// TIA Portal V19 export
FUNCTION "RO_1" : Void   // FC10, LAD
{ S7_Optimized_Access := 'TRUE' }
// stored: SetENOAutomatically false
   VAR_TEMP   // added for the SCL form of the ladder/FBD networks
      _w1 : Bool;
      _w2 : Bool;
      _w3 : Bool;
   END_VAR
BEGIN

REGION Network 1: ABV-301/ ABV-302
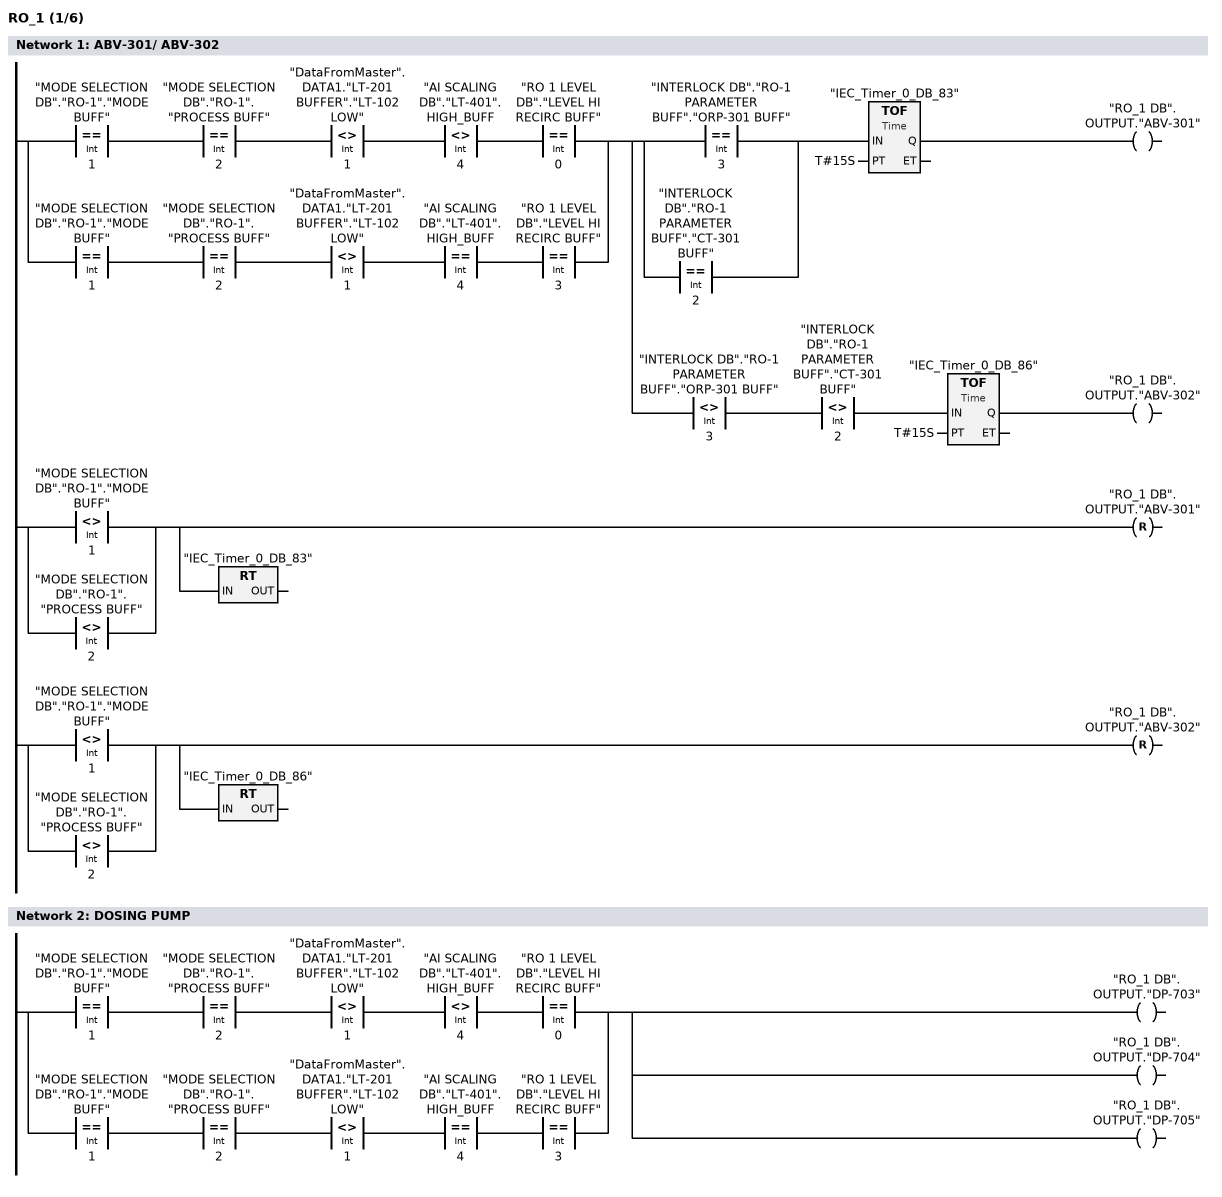
   RUNG wire#powerrail
      { S7_Templates := "SrcType := Int" } EQ_Contact(in1 := "MODE SELECTION DB"."RO-1"."MODE BUFF", in2 := 1)
      { S7_Templates := "SrcType := Int" } EQ_Contact(in1 := "MODE SELECTION DB"."RO-1"."PROCESS BUFF", in2 := 2)
      { S7_Templates := "SrcType := Int" } NE_Contact(in1 := "DataFromMaster".DATA1."LT-201 BUFFER"."LT-102 LOW", in2 := 1)
      { S7_Templates := "SrcType := Int" } NE_Contact(in1 := "AI SCALING DB"."LT-401".HIGH_BUFF, in2 := 4)
      { S7_Templates := "SrcType := Int" } EQ_Contact(in1 := "RO 1 LEVEL DB"."LEVEL HI RECIRC BUFF", in2 := 0)
      wire#w1
      { S7_Templates := "SrcType := Int" } EQ_Contact(in1 := "INTERLOCK DB"."RO-1 PARAMETER BUFF"."ORP-301 BUFF", in2 := 3)
      wire#w2
      { S7_Templates := "time_type := Time" } "IEC_Timer_0_DB_83".TOF(pt := T#15S, et =>)
      Coil( "RO_1 DB".OUTPUT."ABV-301" )
   END_RUNG
   RUNG wire#powerrail
      { S7_Templates := "SrcType := Int" } EQ_Contact(in1 := "MODE SELECTION DB"."RO-1"."MODE BUFF", in2 := 1)
      { S7_Templates := "SrcType := Int" } EQ_Contact(in1 := "MODE SELECTION DB"."RO-1"."PROCESS BUFF", in2 := 2)
      { S7_Templates := "SrcType := Int" } NE_Contact(in1 := "DataFromMaster".DATA1."LT-201 BUFFER"."LT-102 LOW", in2 := 1)
      { S7_Templates := "SrcType := Int" } EQ_Contact(in1 := "AI SCALING DB"."LT-401".HIGH_BUFF, in2 := 4)
      { S7_Templates := "SrcType := Int" } EQ_Contact(in1 := "RO 1 LEVEL DB"."LEVEL HI RECIRC BUFF", in2 := 3)
   END_RUNG wire#w1
   RUNG wire#w1
      { S7_Templates := "SrcType := Int" } EQ_Contact(in1 := "INTERLOCK DB"."RO-1 PARAMETER BUFF"."CT-301 BUFF", in2 := 2)
   END_RUNG wire#w2
   RUNG wire#w1
      { S7_Templates := "SrcType := Int" } NE_Contact(in1 := "INTERLOCK DB"."RO-1 PARAMETER BUFF"."ORP-301 BUFF", in2 := 3)
      { S7_Templates := "SrcType := Int" } NE_Contact(in1 := "INTERLOCK DB"."RO-1 PARAMETER BUFF"."CT-301 BUFF", in2 := 2)
      { S7_Templates := "time_type := Time" } "IEC_Timer_0_DB_86".TOF(pt := T#15S, et =>)
      Coil( "RO_1 DB".OUTPUT."ABV-302" )
   END_RUNG
   RUNG wire#powerrail
      { S7_Templates := "SrcType := Int" } NE_Contact(in1 := "MODE SELECTION DB"."RO-1"."MODE BUFF", in2 := 1)
      wire#w3
      R_Coil( "RO_1 DB".OUTPUT."ABV-301" )
   END_RUNG
   RUNG wire#powerrail
      { S7_Templates := "SrcType := Int" } NE_Contact(in1 := "MODE SELECTION DB"."RO-1"."PROCESS BUFF", in2 := 2)
   END_RUNG wire#w3
   RUNG wire#w3
      RT_Coil( "IEC_Timer_0_DB_83" )
   END_RUNG
   RUNG wire#powerrail
      { S7_Templates := "SrcType := Int" } NE_Contact(in1 := "MODE SELECTION DB"."RO-1"."MODE BUFF", in2 := 1)
      wire#w4
      R_Coil( "RO_1 DB".OUTPUT."ABV-302" )
   END_RUNG
   RUNG wire#powerrail
      { S7_Templates := "SrcType := Int" } NE_Contact(in1 := "MODE SELECTION DB"."RO-1"."PROCESS BUFF", in2 := 2)
   END_RUNG wire#w4
   RUNG wire#w4
      RT_Coil( "IEC_Timer_0_DB_86" )
   END_RUNG
   // the same network as SCL:
   #_w1 := (("MODE SELECTION DB"."RO-1"."MODE BUFF" = 1) AND ("MODE SELECTION DB"."RO-1"."PROCESS BUFF" = 2) AND ("DataFromMaster".DATA1."LT-201 BUFFER"."LT-102 LOW" <> 1) AND ("AI SCALING DB"."LT-401".HIGH_BUFF <> 4) AND ("RO 1 LEVEL DB"."LEVEL HI RECIRC BUFF" = 0)) OR (("MODE SELECTION DB"."RO-1"."MODE BUFF" = 1) AND ("MODE SELECTION DB"."RO-1"."PROCESS BUFF" = 2) AND ("DataFromMaster".DATA1."LT-201 BUFFER"."LT-102 LOW" <> 1) AND ("AI SCALING DB"."LT-401".HIGH_BUFF = 4) AND ("RO 1 LEVEL DB"."LEVEL HI RECIRC BUFF" = 3));
   "IEC_Timer_0_DB_83".TOF(IN := #_w1 AND (("INTERLOCK DB"."RO-1 PARAMETER BUFF"."ORP-301 BUFF" = 3) OR ("INTERLOCK DB"."RO-1 PARAMETER BUFF"."CT-301 BUFF" = 2)),
                           PT := T#15S);
   "RO_1 DB".OUTPUT."ABV-301" := "IEC_Timer_0_DB_83".Q;
   "IEC_Timer_0_DB_86".TOF(IN := #_w1 AND ("INTERLOCK DB"."RO-1 PARAMETER BUFF"."ORP-301 BUFF" <> 3) AND ("INTERLOCK DB"."RO-1 PARAMETER BUFF"."CT-301 BUFF" <> 2),
                           PT := T#15S);
   "RO_1 DB".OUTPUT."ABV-302" := "IEC_Timer_0_DB_86".Q;
   #_w2 := ("MODE SELECTION DB"."RO-1"."MODE BUFF" <> 1) OR ("MODE SELECTION DB"."RO-1"."PROCESS BUFF" <> 2);
   IF #_w2 THEN
       "RO_1 DB".OUTPUT."ABV-301" := FALSE;
       RESET_TIMER("IEC_Timer_0_DB_83");
   END_IF;
   #_w3 := ("MODE SELECTION DB"."RO-1"."MODE BUFF" <> 1) OR ("MODE SELECTION DB"."RO-1"."PROCESS BUFF" <> 2);
   IF #_w3 THEN
       "RO_1 DB".OUTPUT."ABV-302" := FALSE;
       RESET_TIMER("IEC_Timer_0_DB_86");
   END_IF;
END_REGION

REGION Network 2: DOSING PUMP
   RUNG wire#powerrail
      { S7_Templates := "SrcType := Int" } EQ_Contact(in1 := "MODE SELECTION DB"."RO-1"."MODE BUFF", in2 := 1)
      { S7_Templates := "SrcType := Int" } EQ_Contact(in1 := "MODE SELECTION DB"."RO-1"."PROCESS BUFF", in2 := 2)
      { S7_Templates := "SrcType := Int" } NE_Contact(in1 := "DataFromMaster".DATA1."LT-201 BUFFER"."LT-102 LOW", in2 := 1)
      { S7_Templates := "SrcType := Int" } NE_Contact(in1 := "AI SCALING DB"."LT-401".HIGH_BUFF, in2 := 4)
      { S7_Templates := "SrcType := Int" } EQ_Contact(in1 := "RO 1 LEVEL DB"."LEVEL HI RECIRC BUFF", in2 := 0)
      wire#w1
      Coil( "RO_1 DB".OUTPUT."DP-703" )
   END_RUNG
   RUNG wire#powerrail
      { S7_Templates := "SrcType := Int" } EQ_Contact(in1 := "MODE SELECTION DB"."RO-1"."MODE BUFF", in2 := 1)
      { S7_Templates := "SrcType := Int" } EQ_Contact(in1 := "MODE SELECTION DB"."RO-1"."PROCESS BUFF", in2 := 2)
      { S7_Templates := "SrcType := Int" } NE_Contact(in1 := "DataFromMaster".DATA1."LT-201 BUFFER"."LT-102 LOW", in2 := 1)
      { S7_Templates := "SrcType := Int" } EQ_Contact(in1 := "AI SCALING DB"."LT-401".HIGH_BUFF, in2 := 4)
      { S7_Templates := "SrcType := Int" } EQ_Contact(in1 := "RO 1 LEVEL DB"."LEVEL HI RECIRC BUFF", in2 := 3)
   END_RUNG wire#w1
   RUNG wire#w1
      Coil( "RO_1 DB".OUTPUT."DP-704" )
   END_RUNG
   RUNG wire#w1
      Coil( "RO_1 DB".OUTPUT."DP-705" )
   END_RUNG
   // the same network as SCL:
   "RO_1 DB".OUTPUT."DP-703" := (("MODE SELECTION DB"."RO-1"."MODE BUFF" = 1) AND ("MODE SELECTION DB"."RO-1"."PROCESS BUFF" = 2) AND ("DataFromMaster".DATA1."LT-201 BUFFER"."LT-102 LOW" <> 1) AND ("AI SCALING DB"."LT-401".HIGH_BUFF <> 4) AND ("RO 1 LEVEL DB"."LEVEL HI RECIRC BUFF" = 0)) OR (("MODE SELECTION DB"."RO-1"."MODE BUFF" = 1) AND ("MODE SELECTION DB"."RO-1"."PROCESS BUFF" = 2) AND ("DataFromMaster".DATA1."LT-201 BUFFER"."LT-102 LOW" <> 1) AND ("AI SCALING DB"."LT-401".HIGH_BUFF = 4) AND ("RO 1 LEVEL DB"."LEVEL HI RECIRC BUFF" = 3));
   "RO_1 DB".OUTPUT."DP-704" := "RO_1 DB".OUTPUT."DP-703";
   "RO_1 DB".OUTPUT."DP-705" := "RO_1 DB".OUTPUT."DP-703";
END_REGION

REGION Network 3: RO-1 FEED PUMP
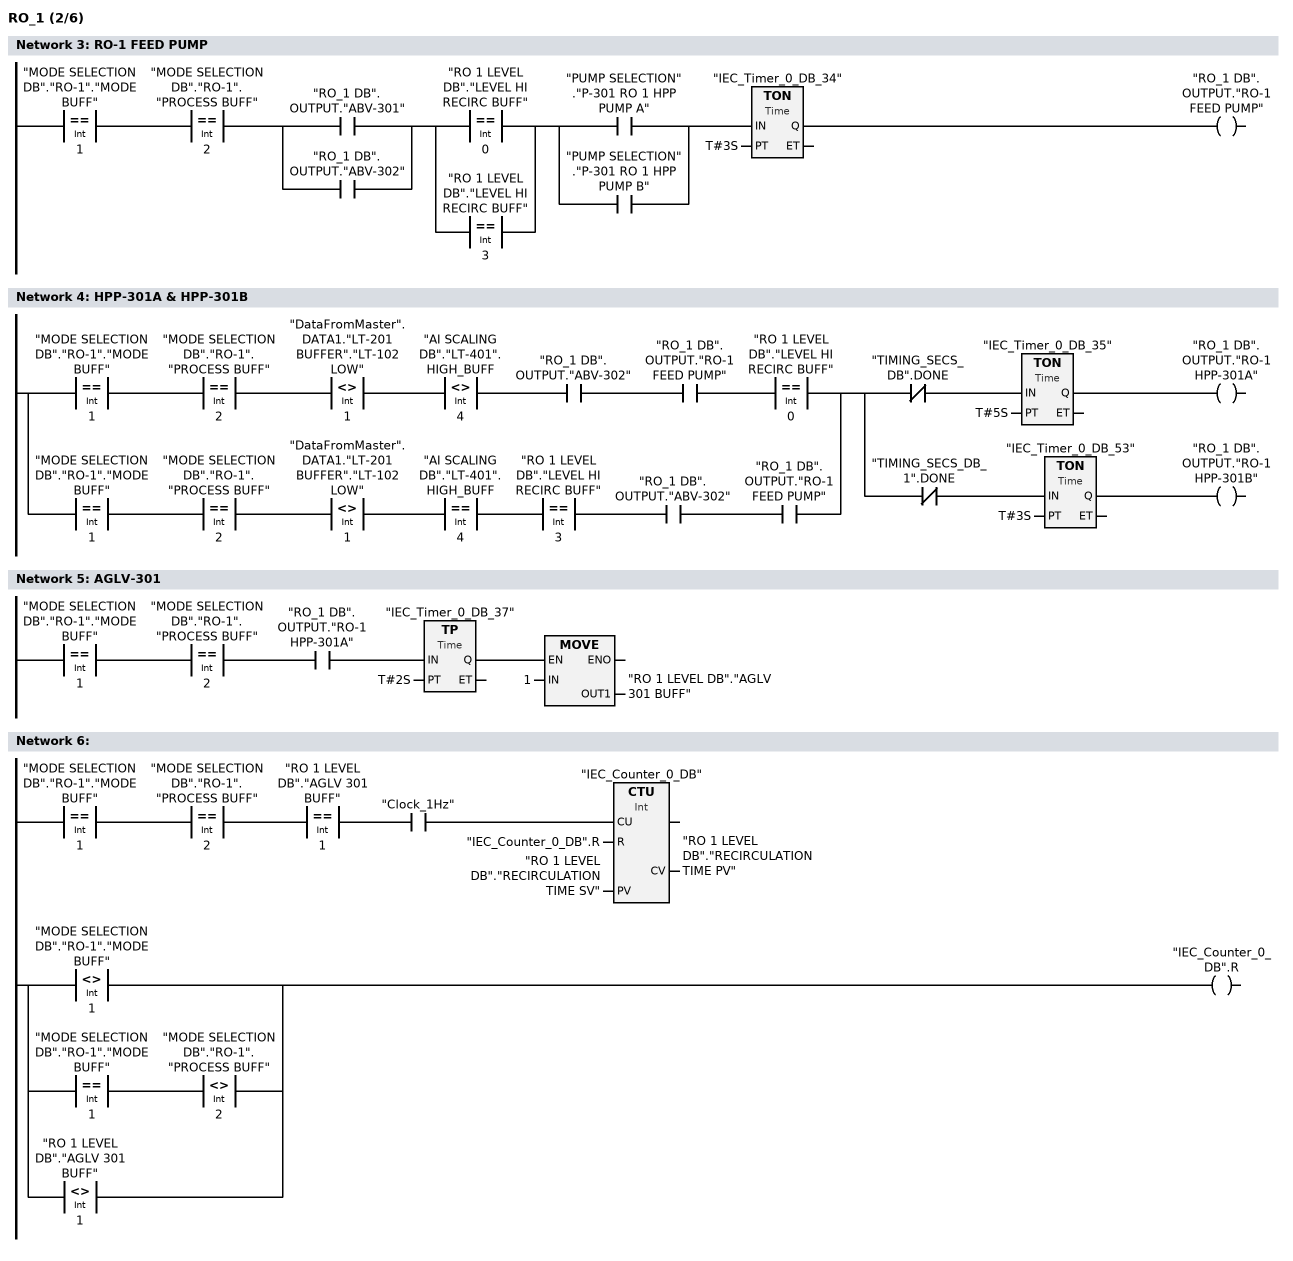
   RUNG wire#powerrail
      { S7_Templates := "SrcType := Int" } EQ_Contact(in1 := "MODE SELECTION DB"."RO-1"."MODE BUFF", in2 := 1)
      { S7_Templates := "SrcType := Int" } EQ_Contact(in1 := "MODE SELECTION DB"."RO-1"."PROCESS BUFF", in2 := 2)
      wire#w1
      Contact( "RO_1 DB".OUTPUT."ABV-301" )
      wire#w2
      { S7_Templates := "SrcType := Int" } EQ_Contact(in1 := "RO 1 LEVEL DB"."LEVEL HI RECIRC BUFF", in2 := 0)
      wire#w3
      Contact( "PUMP SELECTION"."P-301 RO 1 HPP PUMP A" )
      wire#w4
      { S7_Templates := "time_type := Time" } "IEC_Timer_0_DB_34".TON(pt := T#3S, et =>)
      Coil( "RO_1 DB".OUTPUT."RO-1 FEED PUMP" )
   END_RUNG
   RUNG wire#w1
      Contact( "RO_1 DB".OUTPUT."ABV-302" )
   END_RUNG wire#w2
   RUNG wire#w2
      { S7_Templates := "SrcType := Int" } EQ_Contact(in1 := "RO 1 LEVEL DB"."LEVEL HI RECIRC BUFF", in2 := 3)
   END_RUNG wire#w3
   RUNG wire#w3
      Contact( "PUMP SELECTION"."P-301 RO 1 HPP PUMP B" )
   END_RUNG wire#w4
   // the same network as SCL:
   "IEC_Timer_0_DB_34".TON(IN := ("MODE SELECTION DB"."RO-1"."MODE BUFF" = 1) AND ("MODE SELECTION DB"."RO-1"."PROCESS BUFF" = 2) AND ("RO_1 DB".OUTPUT."ABV-301" OR "RO_1 DB".OUTPUT."ABV-302") AND (("RO 1 LEVEL DB"."LEVEL HI RECIRC BUFF" = 0) OR ("RO 1 LEVEL DB"."LEVEL HI RECIRC BUFF" = 3)) AND ("PUMP SELECTION"."P-301 RO 1 HPP PUMP A" OR "PUMP SELECTION"."P-301 RO 1 HPP PUMP B"),
                           PT := T#3S);
   "RO_1 DB".OUTPUT."RO-1 FEED PUMP" := "IEC_Timer_0_DB_34".Q;
END_REGION

REGION Network 4: HPP-301A & HPP-301B
   RUNG wire#powerrail
      { S7_Templates := "SrcType := Int" } EQ_Contact(in1 := "MODE SELECTION DB"."RO-1"."MODE BUFF", in2 := 1)
      { S7_Templates := "SrcType := Int" } EQ_Contact(in1 := "MODE SELECTION DB"."RO-1"."PROCESS BUFF", in2 := 2)
      { S7_Templates := "SrcType := Int" } NE_Contact(in1 := "DataFromMaster".DATA1."LT-201 BUFFER"."LT-102 LOW", in2 := 1)
      { S7_Templates := "SrcType := Int" } NE_Contact(in1 := "AI SCALING DB"."LT-401".HIGH_BUFF, in2 := 4)
      Contact( "RO_1 DB".OUTPUT."ABV-302" )
      Contact( "RO_1 DB".OUTPUT."RO-1 FEED PUMP" )
      { S7_Templates := "SrcType := Int" } EQ_Contact(in1 := "RO 1 LEVEL DB"."LEVEL HI RECIRC BUFF", in2 := 0)
      wire#w1
      I_Contact( "TIMING_SECS_DB".DONE )
      { S7_Templates := "time_type := Time" } "IEC_Timer_0_DB_35".TON(pt := T#5S, et =>)
      Coil( "RO_1 DB".OUTPUT."RO-1 HPP-301A" )
   END_RUNG
   RUNG wire#powerrail
      { S7_Templates := "SrcType := Int" } EQ_Contact(in1 := "MODE SELECTION DB"."RO-1"."MODE BUFF", in2 := 1)
      { S7_Templates := "SrcType := Int" } EQ_Contact(in1 := "MODE SELECTION DB"."RO-1"."PROCESS BUFF", in2 := 2)
      { S7_Templates := "SrcType := Int" } NE_Contact(in1 := "DataFromMaster".DATA1."LT-201 BUFFER"."LT-102 LOW", in2 := 1)
      { S7_Templates := "SrcType := Int" } EQ_Contact(in1 := "AI SCALING DB"."LT-401".HIGH_BUFF, in2 := 4)
      { S7_Templates := "SrcType := Int" } EQ_Contact(in1 := "RO 1 LEVEL DB"."LEVEL HI RECIRC BUFF", in2 := 3)
      Contact( "RO_1 DB".OUTPUT."ABV-302" )
      Contact( "RO_1 DB".OUTPUT."RO-1 FEED PUMP" )
   END_RUNG wire#w1
   RUNG wire#w1
      I_Contact( "TIMING_SECS_DB_1".DONE )
      { S7_Templates := "time_type := Time" } "IEC_Timer_0_DB_53".TON(pt := T#3S, et =>)
      Coil( "RO_1 DB".OUTPUT."RO-1 HPP-301B" )
   END_RUNG
   // the same network as SCL:
   #_w1 := (("MODE SELECTION DB"."RO-1"."MODE BUFF" = 1) AND ("MODE SELECTION DB"."RO-1"."PROCESS BUFF" = 2) AND ("DataFromMaster".DATA1."LT-201 BUFFER"."LT-102 LOW" <> 1) AND ("AI SCALING DB"."LT-401".HIGH_BUFF <> 4) AND "RO_1 DB".OUTPUT."ABV-302" AND "RO_1 DB".OUTPUT."RO-1 FEED PUMP" AND ("RO 1 LEVEL DB"."LEVEL HI RECIRC BUFF" = 0)) OR (("MODE SELECTION DB"."RO-1"."MODE BUFF" = 1) AND ("MODE SELECTION DB"."RO-1"."PROCESS BUFF" = 2) AND ("DataFromMaster".DATA1."LT-201 BUFFER"."LT-102 LOW" <> 1) AND ("AI SCALING DB"."LT-401".HIGH_BUFF = 4) AND ("RO 1 LEVEL DB"."LEVEL HI RECIRC BUFF" = 3) AND "RO_1 DB".OUTPUT."ABV-302" AND "RO_1 DB".OUTPUT."RO-1 FEED PUMP");
   "IEC_Timer_0_DB_35".TON(IN := #_w1 AND NOT "TIMING_SECS_DB".DONE, PT := T#5S);
   "RO_1 DB".OUTPUT."RO-1 HPP-301A" := "IEC_Timer_0_DB_35".Q;
   "IEC_Timer_0_DB_53".TON(IN := #_w1 AND NOT "TIMING_SECS_DB_1".DONE, PT := T#3S);
   "RO_1 DB".OUTPUT."RO-1 HPP-301B" := "IEC_Timer_0_DB_53".Q;
END_REGION

REGION Network 5: AGLV-301
   RUNG wire#powerrail
      { S7_Templates := "SrcType := Int" } EQ_Contact(in1 := "MODE SELECTION DB"."RO-1"."MODE BUFF", in2 := 1)
      { S7_Templates := "SrcType := Int" } EQ_Contact(in1 := "MODE SELECTION DB"."RO-1"."PROCESS BUFF", in2 := 2)
      Contact( "RO_1 DB".OUTPUT."RO-1 HPP-301A" )
      { S7_Templates := "time_type := Time" } "IEC_Timer_0_DB_37".TP(pt := T#2S, et =>)
      Move(in := 1, out1 => "RO 1 LEVEL DB"."AGLV 301 BUFF")
   END_RUNG
   // the same network as SCL:
   "IEC_Timer_0_DB_37".TP(IN := ("MODE SELECTION DB"."RO-1"."MODE BUFF" = 1) AND ("MODE SELECTION DB"."RO-1"."PROCESS BUFF" = 2) AND "RO_1 DB".OUTPUT."RO-1 HPP-301A",
                          PT := T#2S);
   IF "IEC_Timer_0_DB_37".Q THEN "RO 1 LEVEL DB"."AGLV 301 BUFF" := 1; END_IF;
END_REGION

REGION Network 6
   RUNG wire#powerrail
      { S7_Templates := "SrcType := Int" } EQ_Contact(in1 := "MODE SELECTION DB"."RO-1"."MODE BUFF", in2 := 1)
      { S7_Templates := "SrcType := Int" } EQ_Contact(in1 := "MODE SELECTION DB"."RO-1"."PROCESS BUFF", in2 := 2)
      { S7_Templates := "SrcType := Int" } EQ_Contact(in1 := "RO 1 LEVEL DB"."AGLV 301 BUFF", in2 := 1)
      Contact( "Clock_1Hz" )
      { S7_Templates := "value_type := Int" } "IEC_Counter_0_DB".CTU(r := "IEC_Counter_0_DB".R, pv := "RO 1 LEVEL DB"."RECIRCULATION TIME SV", cv => "RO 1 LEVEL DB"."RECIRCULATION TIME PV")
   END_RUNG
   RUNG wire#powerrail
      { S7_Templates := "SrcType := Int" } NE_Contact(in1 := "MODE SELECTION DB"."RO-1"."MODE BUFF", in2 := 1)
      wire#w1
      Coil( "IEC_Counter_0_DB".R )
   END_RUNG
   RUNG wire#powerrail
      { S7_Templates := "SrcType := Int" } EQ_Contact(in1 := "MODE SELECTION DB"."RO-1"."MODE BUFF", in2 := 1)
      { S7_Templates := "SrcType := Int" } NE_Contact(in1 := "MODE SELECTION DB"."RO-1"."PROCESS BUFF", in2 := 2)
   END_RUNG wire#w1
   RUNG wire#powerrail
      { S7_Templates := "SrcType := Int" } NE_Contact(in1 := "RO 1 LEVEL DB"."AGLV 301 BUFF", in2 := 1)
   END_RUNG wire#w1
   // the same network as SCL:
   "IEC_Counter_0_DB".CTU(CU := ("MODE SELECTION DB"."RO-1"."MODE BUFF" = 1) AND ("MODE SELECTION DB"."RO-1"."PROCESS BUFF" = 2) AND ("RO 1 LEVEL DB"."AGLV 301 BUFF" = 1) AND "Clock_1Hz",
                          R := "IEC_Counter_0_DB".R,
                          PV := "RO 1 LEVEL DB"."RECIRCULATION TIME SV",
                          CV => "RO 1 LEVEL DB"."RECIRCULATION TIME PV");
   "IEC_Counter_0_DB".R := ("MODE SELECTION DB"."RO-1"."MODE BUFF" <> 1) OR (("MODE SELECTION DB"."RO-1"."MODE BUFF" = 1) AND ("MODE SELECTION DB"."RO-1"."PROCESS BUFF" <> 2)) OR ("RO 1 LEVEL DB"."AGLV 301 BUFF" <> 1);
END_REGION

REGION Network 7
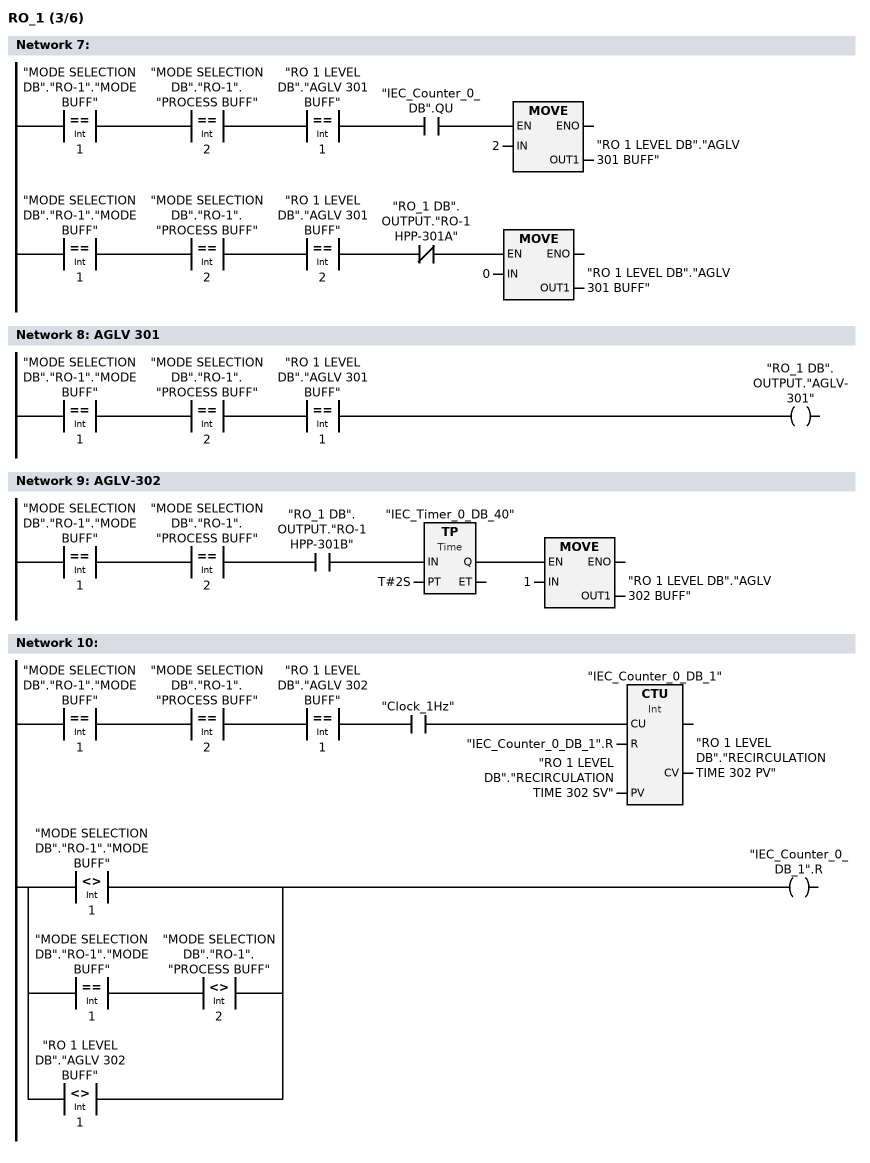
   RUNG wire#powerrail
      { S7_Templates := "SrcType := Int" } EQ_Contact(in1 := "MODE SELECTION DB"."RO-1"."MODE BUFF", in2 := 1)
      { S7_Templates := "SrcType := Int" } EQ_Contact(in1 := "MODE SELECTION DB"."RO-1"."PROCESS BUFF", in2 := 2)
      { S7_Templates := "SrcType := Int" } EQ_Contact(in1 := "RO 1 LEVEL DB"."AGLV 301 BUFF", in2 := 1)
      Contact( "IEC_Counter_0_DB".QU )
      Move(in := 2, out1 => "RO 1 LEVEL DB"."AGLV 301 BUFF")
   END_RUNG
   RUNG wire#powerrail
      { S7_Templates := "SrcType := Int" } EQ_Contact(in1 := "MODE SELECTION DB"."RO-1"."MODE BUFF", in2 := 1)
      { S7_Templates := "SrcType := Int" } EQ_Contact(in1 := "MODE SELECTION DB"."RO-1"."PROCESS BUFF", in2 := 2)
      { S7_Templates := "SrcType := Int" } EQ_Contact(in1 := "RO 1 LEVEL DB"."AGLV 301 BUFF", in2 := 2)
      I_Contact( "RO_1 DB".OUTPUT."RO-1 HPP-301A" )
      Move(in := 0, out1 => "RO 1 LEVEL DB"."AGLV 301 BUFF")
   END_RUNG
   // the same network as SCL:
   IF ("MODE SELECTION DB"."RO-1"."MODE BUFF" = 1) AND ("MODE SELECTION DB"."RO-1"."PROCESS BUFF" = 2) AND ("RO 1 LEVEL DB"."AGLV 301 BUFF" = 1) AND "IEC_Counter_0_DB".QU THEN
       "RO 1 LEVEL DB"."AGLV 301 BUFF" := 2;
   END_IF;
   IF ("MODE SELECTION DB"."RO-1"."MODE BUFF" = 1) AND ("MODE SELECTION DB"."RO-1"."PROCESS BUFF" = 2) AND ("RO 1 LEVEL DB"."AGLV 301 BUFF" = 2) AND NOT "RO_1 DB".OUTPUT."RO-1 HPP-301A" THEN
       "RO 1 LEVEL DB"."AGLV 301 BUFF" := 0;
   END_IF;
END_REGION

REGION Network 8: AGLV 301
   RUNG wire#powerrail
      { S7_Templates := "SrcType := Int" } EQ_Contact(in1 := "MODE SELECTION DB"."RO-1"."MODE BUFF", in2 := 1)
      { S7_Templates := "SrcType := Int" } EQ_Contact(in1 := "MODE SELECTION DB"."RO-1"."PROCESS BUFF", in2 := 2)
      { S7_Templates := "SrcType := Int" } EQ_Contact(in1 := "RO 1 LEVEL DB"."AGLV 301 BUFF", in2 := 1)
      Coil( "RO_1 DB".OUTPUT."AGLV-301" )
   END_RUNG
   // the same network as SCL:
   "RO_1 DB".OUTPUT."AGLV-301" := ("MODE SELECTION DB"."RO-1"."MODE BUFF" = 1) AND ("MODE SELECTION DB"."RO-1"."PROCESS BUFF" = 2) AND ("RO 1 LEVEL DB"."AGLV 301 BUFF" = 1);
END_REGION

REGION Network 9: AGLV-302
   RUNG wire#powerrail
      { S7_Templates := "SrcType := Int" } EQ_Contact(in1 := "MODE SELECTION DB"."RO-1"."MODE BUFF", in2 := 1)
      { S7_Templates := "SrcType := Int" } EQ_Contact(in1 := "MODE SELECTION DB"."RO-1"."PROCESS BUFF", in2 := 2)
      Contact( "RO_1 DB".OUTPUT."RO-1 HPP-301B" )
      { S7_Templates := "time_type := Time" } "IEC_Timer_0_DB_40".TP(pt := T#2S, et =>)
      Move(in := 1, out1 => "RO 1 LEVEL DB"."AGLV 302 BUFF")
   END_RUNG
   // the same network as SCL:
   "IEC_Timer_0_DB_40".TP(IN := ("MODE SELECTION DB"."RO-1"."MODE BUFF" = 1) AND ("MODE SELECTION DB"."RO-1"."PROCESS BUFF" = 2) AND "RO_1 DB".OUTPUT."RO-1 HPP-301B",
                          PT := T#2S);
   IF "IEC_Timer_0_DB_40".Q THEN "RO 1 LEVEL DB"."AGLV 302 BUFF" := 1; END_IF;
END_REGION

REGION Network 10
   RUNG wire#powerrail
      { S7_Templates := "SrcType := Int" } EQ_Contact(in1 := "MODE SELECTION DB"."RO-1"."MODE BUFF", in2 := 1)
      { S7_Templates := "SrcType := Int" } EQ_Contact(in1 := "MODE SELECTION DB"."RO-1"."PROCESS BUFF", in2 := 2)
      { S7_Templates := "SrcType := Int" } EQ_Contact(in1 := "RO 1 LEVEL DB"."AGLV 302 BUFF", in2 := 1)
      Contact( "Clock_1Hz" )
      { S7_Templates := "value_type := Int" } "IEC_Counter_0_DB_1".CTU(r := "IEC_Counter_0_DB_1".R, pv := "RO 1 LEVEL DB"."RECIRCULATION TIME 302 SV", cv => "RO 1 LEVEL DB"."RECIRCULATION TIME 302 PV")
   END_RUNG
   RUNG wire#powerrail
      { S7_Templates := "SrcType := Int" } NE_Contact(in1 := "MODE SELECTION DB"."RO-1"."MODE BUFF", in2 := 1)
      wire#w1
      Coil( "IEC_Counter_0_DB_1".R )
   END_RUNG
   RUNG wire#powerrail
      { S7_Templates := "SrcType := Int" } EQ_Contact(in1 := "MODE SELECTION DB"."RO-1"."MODE BUFF", in2 := 1)
      { S7_Templates := "SrcType := Int" } NE_Contact(in1 := "MODE SELECTION DB"."RO-1"."PROCESS BUFF", in2 := 2)
   END_RUNG wire#w1
   RUNG wire#powerrail
      { S7_Templates := "SrcType := Int" } NE_Contact(in1 := "RO 1 LEVEL DB"."AGLV 302 BUFF", in2 := 1)
   END_RUNG wire#w1
   // the same network as SCL:
   "IEC_Counter_0_DB_1".CTU(CU := ("MODE SELECTION DB"."RO-1"."MODE BUFF" = 1) AND ("MODE SELECTION DB"."RO-1"."PROCESS BUFF" = 2) AND ("RO 1 LEVEL DB"."AGLV 302 BUFF" = 1) AND "Clock_1Hz",
                           R := "IEC_Counter_0_DB_1".R,
                           PV := "RO 1 LEVEL DB"."RECIRCULATION TIME 302 SV",
                           CV => "RO 1 LEVEL DB"."RECIRCULATION TIME 302 PV");
   "IEC_Counter_0_DB_1".R := ("MODE SELECTION DB"."RO-1"."MODE BUFF" <> 1) OR (("MODE SELECTION DB"."RO-1"."MODE BUFF" = 1) AND ("MODE SELECTION DB"."RO-1"."PROCESS BUFF" <> 2)) OR ("RO 1 LEVEL DB"."AGLV 302 BUFF" <> 1);
END_REGION

REGION Network 11
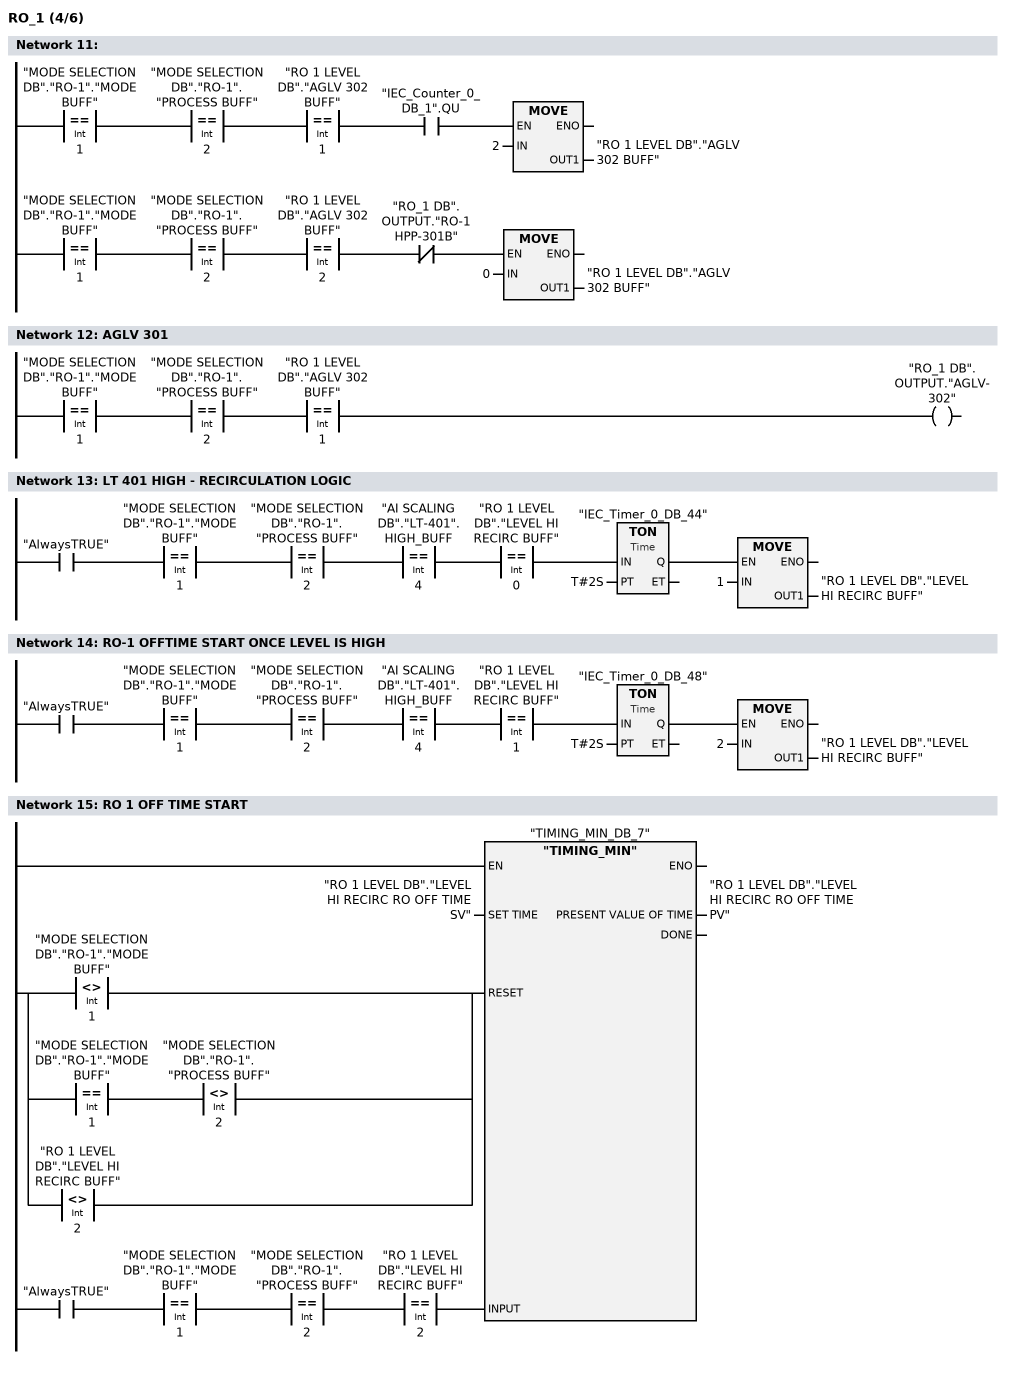
   RUNG wire#powerrail
      { S7_Templates := "SrcType := Int" } EQ_Contact(in1 := "MODE SELECTION DB"."RO-1"."MODE BUFF", in2 := 1)
      { S7_Templates := "SrcType := Int" } EQ_Contact(in1 := "MODE SELECTION DB"."RO-1"."PROCESS BUFF", in2 := 2)
      { S7_Templates := "SrcType := Int" } EQ_Contact(in1 := "RO 1 LEVEL DB"."AGLV 302 BUFF", in2 := 1)
      Contact( "IEC_Counter_0_DB_1".QU )
      Move(in := 2, out1 => "RO 1 LEVEL DB"."AGLV 302 BUFF")
   END_RUNG
   RUNG wire#powerrail
      { S7_Templates := "SrcType := Int" } EQ_Contact(in1 := "MODE SELECTION DB"."RO-1"."MODE BUFF", in2 := 1)
      { S7_Templates := "SrcType := Int" } EQ_Contact(in1 := "MODE SELECTION DB"."RO-1"."PROCESS BUFF", in2 := 2)
      { S7_Templates := "SrcType := Int" } EQ_Contact(in1 := "RO 1 LEVEL DB"."AGLV 302 BUFF", in2 := 2)
      I_Contact( "RO_1 DB".OUTPUT."RO-1 HPP-301B" )
      Move(in := 0, out1 => "RO 1 LEVEL DB"."AGLV 302 BUFF")
   END_RUNG
   // the same network as SCL:
   IF ("MODE SELECTION DB"."RO-1"."MODE BUFF" = 1) AND ("MODE SELECTION DB"."RO-1"."PROCESS BUFF" = 2) AND ("RO 1 LEVEL DB"."AGLV 302 BUFF" = 1) AND "IEC_Counter_0_DB_1".QU THEN
       "RO 1 LEVEL DB"."AGLV 302 BUFF" := 2;
   END_IF;
   IF ("MODE SELECTION DB"."RO-1"."MODE BUFF" = 1) AND ("MODE SELECTION DB"."RO-1"."PROCESS BUFF" = 2) AND ("RO 1 LEVEL DB"."AGLV 302 BUFF" = 2) AND NOT "RO_1 DB".OUTPUT."RO-1 HPP-301B" THEN
       "RO 1 LEVEL DB"."AGLV 302 BUFF" := 0;
   END_IF;
END_REGION

REGION Network 12: AGLV 301
   RUNG wire#powerrail
      { S7_Templates := "SrcType := Int" } EQ_Contact(in1 := "MODE SELECTION DB"."RO-1"."MODE BUFF", in2 := 1)
      { S7_Templates := "SrcType := Int" } EQ_Contact(in1 := "MODE SELECTION DB"."RO-1"."PROCESS BUFF", in2 := 2)
      { S7_Templates := "SrcType := Int" } EQ_Contact(in1 := "RO 1 LEVEL DB"."AGLV 302 BUFF", in2 := 1)
      Coil( "RO_1 DB".OUTPUT."AGLV-302" )
   END_RUNG
   // the same network as SCL:
   "RO_1 DB".OUTPUT."AGLV-302" := ("MODE SELECTION DB"."RO-1"."MODE BUFF" = 1) AND ("MODE SELECTION DB"."RO-1"."PROCESS BUFF" = 2) AND ("RO 1 LEVEL DB"."AGLV 302 BUFF" = 1);
END_REGION

REGION Network 13: LT 401 HIGH - RECIRCULATION LOGIC
   RUNG wire#powerrail
      Contact( "AlwaysTRUE" )
      { S7_Templates := "SrcType := Int" } EQ_Contact(in1 := "MODE SELECTION DB"."RO-1"."MODE BUFF", in2 := 1)
      { S7_Templates := "SrcType := Int" } EQ_Contact(in1 := "MODE SELECTION DB"."RO-1"."PROCESS BUFF", in2 := 2)
      { S7_Templates := "SrcType := Int" } EQ_Contact(in1 := "AI SCALING DB"."LT-401".HIGH_BUFF, in2 := 4)
      { S7_Templates := "SrcType := Int" } EQ_Contact(in1 := "RO 1 LEVEL DB"."LEVEL HI RECIRC BUFF", in2 := 0)
      { S7_Templates := "time_type := Time" } "IEC_Timer_0_DB_44".TON(pt := T#2S, et =>)
      Move(in := 1, out1 => "RO 1 LEVEL DB"."LEVEL HI RECIRC BUFF")
   END_RUNG
   // the same network as SCL:
   "IEC_Timer_0_DB_44".TON(IN := "AlwaysTRUE" AND ("MODE SELECTION DB"."RO-1"."MODE BUFF" = 1) AND ("MODE SELECTION DB"."RO-1"."PROCESS BUFF" = 2) AND ("AI SCALING DB"."LT-401".HIGH_BUFF = 4) AND ("RO 1 LEVEL DB"."LEVEL HI RECIRC BUFF" = 0),
                           PT := T#2S);
   IF "IEC_Timer_0_DB_44".Q THEN "RO 1 LEVEL DB"."LEVEL HI RECIRC BUFF" := 1; END_IF;
END_REGION

REGION Network 14: RO-1 OFFTIME START ONCE LEVEL IS HIGH
   RUNG wire#powerrail
      Contact( "AlwaysTRUE" )
      { S7_Templates := "SrcType := Int" } EQ_Contact(in1 := "MODE SELECTION DB"."RO-1"."MODE BUFF", in2 := 1)
      { S7_Templates := "SrcType := Int" } EQ_Contact(in1 := "MODE SELECTION DB"."RO-1"."PROCESS BUFF", in2 := 2)
      { S7_Templates := "SrcType := Int" } EQ_Contact(in1 := "AI SCALING DB"."LT-401".HIGH_BUFF, in2 := 4)
      { S7_Templates := "SrcType := Int" } EQ_Contact(in1 := "RO 1 LEVEL DB"."LEVEL HI RECIRC BUFF", in2 := 1)
      { S7_Templates := "time_type := Time" } "IEC_Timer_0_DB_48".TON(pt := T#2S, et =>)
      Move(in := 2, out1 => "RO 1 LEVEL DB"."LEVEL HI RECIRC BUFF")
   END_RUNG
   // the same network as SCL:
   "IEC_Timer_0_DB_48".TON(IN := "AlwaysTRUE" AND ("MODE SELECTION DB"."RO-1"."MODE BUFF" = 1) AND ("MODE SELECTION DB"."RO-1"."PROCESS BUFF" = 2) AND ("AI SCALING DB"."LT-401".HIGH_BUFF = 4) AND ("RO 1 LEVEL DB"."LEVEL HI RECIRC BUFF" = 1),
                           PT := T#2S);
   IF "IEC_Timer_0_DB_48".Q THEN "RO 1 LEVEL DB"."LEVEL HI RECIRC BUFF" := 2; END_IF;
END_REGION

REGION Network 15: RO 1 OFF TIME START
   RUNG wire#powerrail
      "TIMING_MIN_DB_7"(RESET := wire#w1, INPUT := wire#w2, "SET TIME" := "RO 1 LEVEL DB"."LEVEL HI RECIRC RO OFF TIME SV", "PRESENT VALUE OF TIME" => "RO 1 LEVEL DB"."LEVEL HI RECIRC RO OFF TIME PV", DONE =>)
   END_RUNG
   RUNG wire#powerrail
      { S7_Templates := "SrcType := Int" } NE_Contact(in1 := "MODE SELECTION DB"."RO-1"."MODE BUFF", in2 := 1)
   END_RUNG wire#w1
   RUNG wire#powerrail
      { S7_Templates := "SrcType := Int" } EQ_Contact(in1 := "MODE SELECTION DB"."RO-1"."MODE BUFF", in2 := 1)
      { S7_Templates := "SrcType := Int" } NE_Contact(in1 := "MODE SELECTION DB"."RO-1"."PROCESS BUFF", in2 := 2)
   END_RUNG wire#w1
   RUNG wire#powerrail
      { S7_Templates := "SrcType := Int" } NE_Contact(in1 := "RO 1 LEVEL DB"."LEVEL HI RECIRC BUFF", in2 := 2)
   END_RUNG wire#w1
   RUNG wire#powerrail
      Contact( "AlwaysTRUE" )
      { S7_Templates := "SrcType := Int" } EQ_Contact(in1 := "MODE SELECTION DB"."RO-1"."MODE BUFF", in2 := 1)
      { S7_Templates := "SrcType := Int" } EQ_Contact(in1 := "MODE SELECTION DB"."RO-1"."PROCESS BUFF", in2 := 2)
      { S7_Templates := "SrcType := Int" } EQ_Contact(in1 := "RO 1 LEVEL DB"."LEVEL HI RECIRC BUFF", in2 := 2)
   END_RUNG wire#w2
   // the same network as SCL:
   "TIMING_MIN_DB_7"("SET TIME" := "RO 1 LEVEL DB"."LEVEL HI RECIRC RO OFF TIME SV",   // "TIMING_MIN"
                     RESET := ("MODE SELECTION DB"."RO-1"."MODE BUFF" <> 1) OR (("MODE SELECTION DB"."RO-1"."MODE BUFF" = 1) AND ("MODE SELECTION DB"."RO-1"."PROCESS BUFF" <> 2)) OR ("RO 1 LEVEL DB"."LEVEL HI RECIRC BUFF" <> 2),
                     INPUT := "AlwaysTRUE" AND ("MODE SELECTION DB"."RO-1"."MODE BUFF" = 1) AND ("MODE SELECTION DB"."RO-1"."PROCESS BUFF" = 2) AND ("RO 1 LEVEL DB"."LEVEL HI RECIRC BUFF" = 2),
                     "PRESENT VALUE OF TIME" => "RO 1 LEVEL DB"."LEVEL HI RECIRC RO OFF TIME PV");
END_REGION

REGION Network 16: RO 1 RECIRCULATION START AFTER OFF TIME OVER
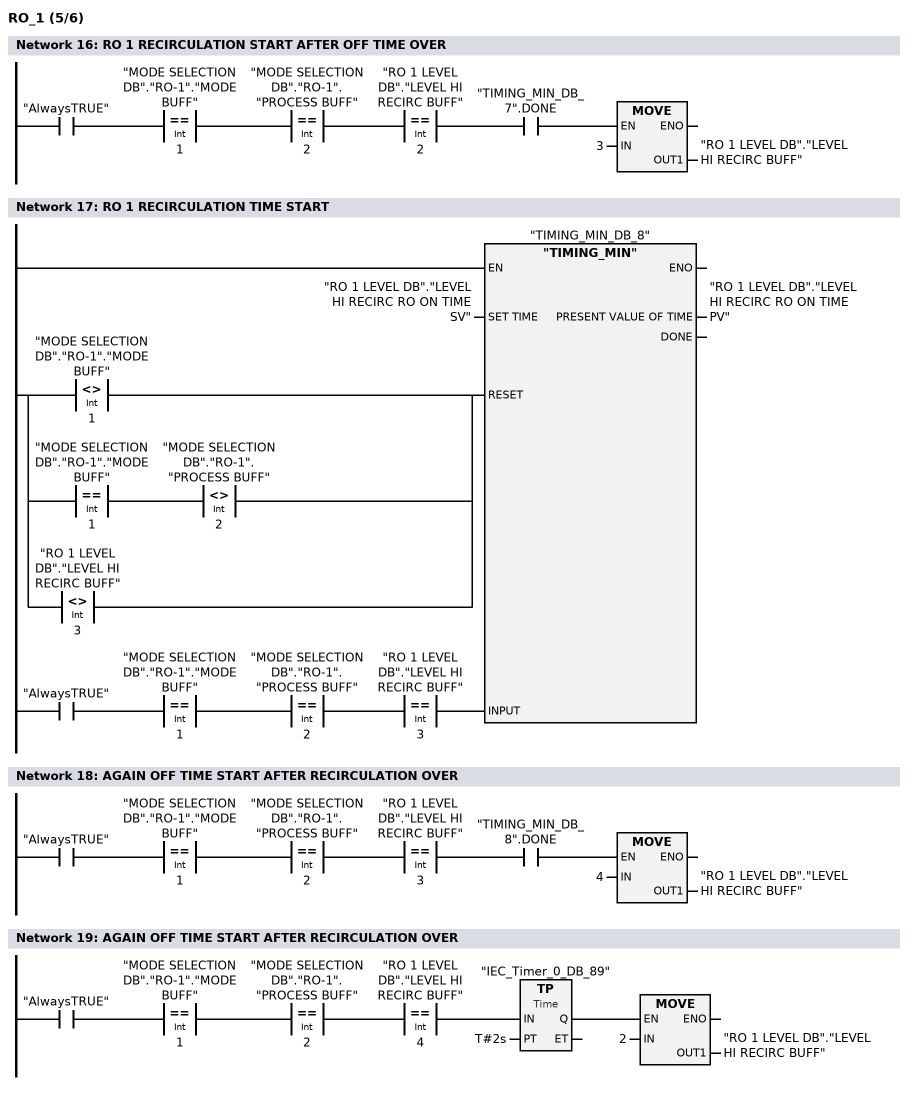
   RUNG wire#powerrail
      Contact( "AlwaysTRUE" )
      { S7_Templates := "SrcType := Int" } EQ_Contact(in1 := "MODE SELECTION DB"."RO-1"."MODE BUFF", in2 := 1)
      { S7_Templates := "SrcType := Int" } EQ_Contact(in1 := "MODE SELECTION DB"."RO-1"."PROCESS BUFF", in2 := 2)
      { S7_Templates := "SrcType := Int" } EQ_Contact(in1 := "RO 1 LEVEL DB"."LEVEL HI RECIRC BUFF", in2 := 2)
      Contact( "TIMING_MIN_DB_7".DONE )
      Move(in := 3, out1 => "RO 1 LEVEL DB"."LEVEL HI RECIRC BUFF")
   END_RUNG
   // the same network as SCL:
   IF "AlwaysTRUE" AND ("MODE SELECTION DB"."RO-1"."MODE BUFF" = 1) AND ("MODE SELECTION DB"."RO-1"."PROCESS BUFF" = 2) AND ("RO 1 LEVEL DB"."LEVEL HI RECIRC BUFF" = 2) AND "TIMING_MIN_DB_7".DONE THEN
       "RO 1 LEVEL DB"."LEVEL HI RECIRC BUFF" := 3;
   END_IF;
END_REGION

REGION Network 17: RO 1 RECIRCULATION TIME START
   RUNG wire#powerrail
      "TIMING_MIN_DB_8"(RESET := wire#w1, INPUT := wire#w2, "SET TIME" := "RO 1 LEVEL DB"."LEVEL HI RECIRC RO ON TIME SV", "PRESENT VALUE OF TIME" => "RO 1 LEVEL DB"."LEVEL HI RECIRC RO ON TIME PV", DONE =>)
   END_RUNG
   RUNG wire#powerrail
      { S7_Templates := "SrcType := Int" } NE_Contact(in1 := "MODE SELECTION DB"."RO-1"."MODE BUFF", in2 := 1)
   END_RUNG wire#w1
   RUNG wire#powerrail
      { S7_Templates := "SrcType := Int" } EQ_Contact(in1 := "MODE SELECTION DB"."RO-1"."MODE BUFF", in2 := 1)
      { S7_Templates := "SrcType := Int" } NE_Contact(in1 := "MODE SELECTION DB"."RO-1"."PROCESS BUFF", in2 := 2)
   END_RUNG wire#w1
   RUNG wire#powerrail
      { S7_Templates := "SrcType := Int" } NE_Contact(in1 := "RO 1 LEVEL DB"."LEVEL HI RECIRC BUFF", in2 := 3)
   END_RUNG wire#w1
   RUNG wire#powerrail
      Contact( "AlwaysTRUE" )
      { S7_Templates := "SrcType := Int" } EQ_Contact(in1 := "MODE SELECTION DB"."RO-1"."MODE BUFF", in2 := 1)
      { S7_Templates := "SrcType := Int" } EQ_Contact(in1 := "MODE SELECTION DB"."RO-1"."PROCESS BUFF", in2 := 2)
      { S7_Templates := "SrcType := Int" } EQ_Contact(in1 := "RO 1 LEVEL DB"."LEVEL HI RECIRC BUFF", in2 := 3)
   END_RUNG wire#w2
   // the same network as SCL:
   "TIMING_MIN_DB_8"("SET TIME" := "RO 1 LEVEL DB"."LEVEL HI RECIRC RO ON TIME SV",   // "TIMING_MIN"
                     RESET := ("MODE SELECTION DB"."RO-1"."MODE BUFF" <> 1) OR (("MODE SELECTION DB"."RO-1"."MODE BUFF" = 1) AND ("MODE SELECTION DB"."RO-1"."PROCESS BUFF" <> 2)) OR ("RO 1 LEVEL DB"."LEVEL HI RECIRC BUFF" <> 3),
                     INPUT := "AlwaysTRUE" AND ("MODE SELECTION DB"."RO-1"."MODE BUFF" = 1) AND ("MODE SELECTION DB"."RO-1"."PROCESS BUFF" = 2) AND ("RO 1 LEVEL DB"."LEVEL HI RECIRC BUFF" = 3),
                     "PRESENT VALUE OF TIME" => "RO 1 LEVEL DB"."LEVEL HI RECIRC RO ON TIME PV");
END_REGION

REGION Network 18: AGAIN OFF TIME START AFTER RECIRCULATION OVER
   RUNG wire#powerrail
      Contact( "AlwaysTRUE" )
      { S7_Templates := "SrcType := Int" } EQ_Contact(in1 := "MODE SELECTION DB"."RO-1"."MODE BUFF", in2 := 1)
      { S7_Templates := "SrcType := Int" } EQ_Contact(in1 := "MODE SELECTION DB"."RO-1"."PROCESS BUFF", in2 := 2)
      { S7_Templates := "SrcType := Int" } EQ_Contact(in1 := "RO 1 LEVEL DB"."LEVEL HI RECIRC BUFF", in2 := 3)
      Contact( "TIMING_MIN_DB_8".DONE )
      Move(in := 4, out1 => "RO 1 LEVEL DB"."LEVEL HI RECIRC BUFF")
   END_RUNG
   // the same network as SCL:
   IF "AlwaysTRUE" AND ("MODE SELECTION DB"."RO-1"."MODE BUFF" = 1) AND ("MODE SELECTION DB"."RO-1"."PROCESS BUFF" = 2) AND ("RO 1 LEVEL DB"."LEVEL HI RECIRC BUFF" = 3) AND "TIMING_MIN_DB_8".DONE THEN
       "RO 1 LEVEL DB"."LEVEL HI RECIRC BUFF" := 4;
   END_IF;
END_REGION

REGION Network 19: AGAIN OFF TIME START AFTER RECIRCULATION OVER
   RUNG wire#powerrail
      Contact( "AlwaysTRUE" )
      { S7_Templates := "SrcType := Int" } EQ_Contact(in1 := "MODE SELECTION DB"."RO-1"."MODE BUFF", in2 := 1)
      { S7_Templates := "SrcType := Int" } EQ_Contact(in1 := "MODE SELECTION DB"."RO-1"."PROCESS BUFF", in2 := 2)
      { S7_Templates := "SrcType := Int" } EQ_Contact(in1 := "RO 1 LEVEL DB"."LEVEL HI RECIRC BUFF", in2 := 4)
      { S7_Templates := "time_type := Time" } "IEC_Timer_0_DB_89".TP(pt := T#2s, et =>)
      Move(in := 2, out1 => "RO 1 LEVEL DB"."LEVEL HI RECIRC BUFF")
   END_RUNG
   // the same network as SCL:
   "IEC_Timer_0_DB_89".TP(IN := "AlwaysTRUE" AND ("MODE SELECTION DB"."RO-1"."MODE BUFF" = 1) AND ("MODE SELECTION DB"."RO-1"."PROCESS BUFF" = 2) AND ("RO 1 LEVEL DB"."LEVEL HI RECIRC BUFF" = 4),
                          PT := T#2s);
   IF "IEC_Timer_0_DB_89".Q THEN "RO 1 LEVEL DB"."LEVEL HI RECIRC BUFF" := 2; END_IF;
END_REGION

REGION Network 20: REcirculation stop when level is normal
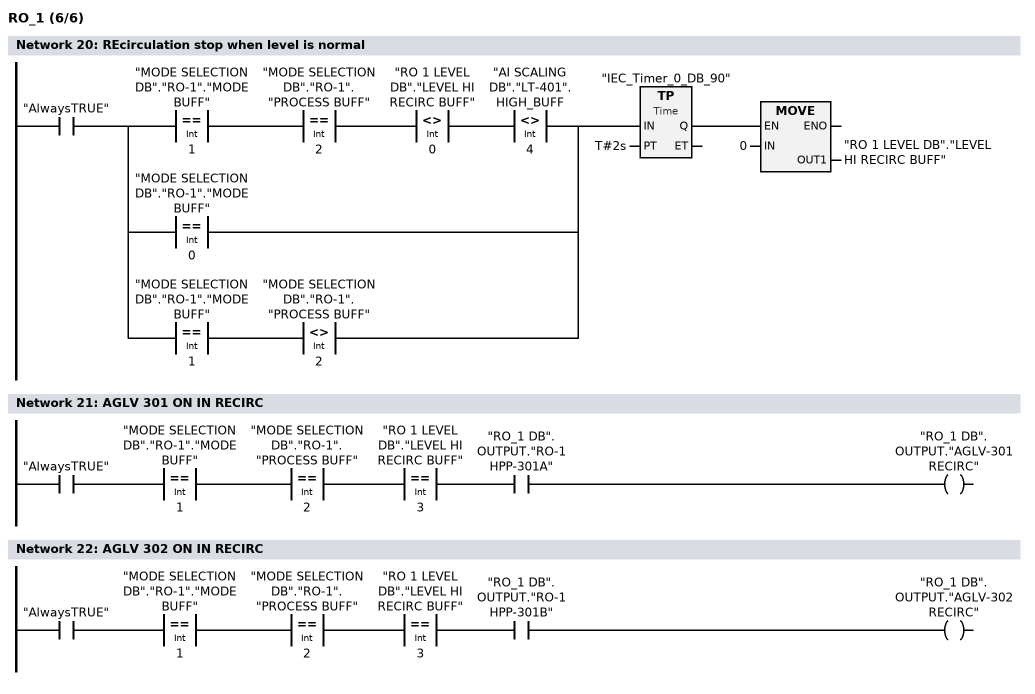
   RUNG wire#powerrail
      Contact( "AlwaysTRUE" )
      wire#w1
      { S7_Templates := "SrcType := Int" } EQ_Contact(in1 := "MODE SELECTION DB"."RO-1"."MODE BUFF", in2 := 1)
      { S7_Templates := "SrcType := Int" } EQ_Contact(in1 := "MODE SELECTION DB"."RO-1"."PROCESS BUFF", in2 := 2)
      { S7_Templates := "SrcType := Int" } NE_Contact(in1 := "RO 1 LEVEL DB"."LEVEL HI RECIRC BUFF", in2 := 0)
      { S7_Templates := "SrcType := Int" } NE_Contact(in1 := "AI SCALING DB"."LT-401".HIGH_BUFF, in2 := 4)
      wire#w2
      { S7_Templates := "time_type := Time" } "IEC_Timer_0_DB_90".TP(pt := T#2s, et =>)
      Move(in := 0, out1 => "RO 1 LEVEL DB"."LEVEL HI RECIRC BUFF")
   END_RUNG
   RUNG wire#w1
      { S7_Templates := "SrcType := Int" } EQ_Contact(in1 := "MODE SELECTION DB"."RO-1"."MODE BUFF", in2 := 0)
   END_RUNG wire#w2
   RUNG wire#w1
      { S7_Templates := "SrcType := Int" } EQ_Contact(in1 := "MODE SELECTION DB"."RO-1"."MODE BUFF", in2 := 1)
      { S7_Templates := "SrcType := Int" } NE_Contact(in1 := "MODE SELECTION DB"."RO-1"."PROCESS BUFF", in2 := 2)
   END_RUNG wire#w2
   // the same network as SCL:
   "IEC_Timer_0_DB_90".TP(IN := "AlwaysTRUE" AND ((("MODE SELECTION DB"."RO-1"."MODE BUFF" = 1) AND ("MODE SELECTION DB"."RO-1"."PROCESS BUFF" = 2) AND ("RO 1 LEVEL DB"."LEVEL HI RECIRC BUFF" <> 0) AND ("AI SCALING DB"."LT-401".HIGH_BUFF <> 4)) OR ("MODE SELECTION DB"."RO-1"."MODE BUFF" = 0) OR (("MODE SELECTION DB"."RO-1"."MODE BUFF" = 1) AND ("MODE SELECTION DB"."RO-1"."PROCESS BUFF" <> 2))),
                          PT := T#2s);
   IF "IEC_Timer_0_DB_90".Q THEN "RO 1 LEVEL DB"."LEVEL HI RECIRC BUFF" := 0; END_IF;
END_REGION

REGION Network 21: AGLV 301 ON IN RECIRC
   RUNG wire#powerrail
      Contact( "AlwaysTRUE" )
      { S7_Templates := "SrcType := Int" } EQ_Contact(in1 := "MODE SELECTION DB"."RO-1"."MODE BUFF", in2 := 1)
      { S7_Templates := "SrcType := Int" } EQ_Contact(in1 := "MODE SELECTION DB"."RO-1"."PROCESS BUFF", in2 := 2)
      { S7_Templates := "SrcType := Int" } EQ_Contact(in1 := "RO 1 LEVEL DB"."LEVEL HI RECIRC BUFF", in2 := 3)
      Contact( "RO_1 DB".OUTPUT."RO-1 HPP-301A" )
      Coil( "RO_1 DB".OUTPUT."AGLV-301 RECIRC" )
   END_RUNG
   // the same network as SCL:
   "RO_1 DB".OUTPUT."AGLV-301 RECIRC" := "AlwaysTRUE" AND ("MODE SELECTION DB"."RO-1"."MODE BUFF" = 1) AND ("MODE SELECTION DB"."RO-1"."PROCESS BUFF" = 2) AND ("RO 1 LEVEL DB"."LEVEL HI RECIRC BUFF" = 3) AND "RO_1 DB".OUTPUT."RO-1 HPP-301A";
END_REGION

REGION Network 22: AGLV 302 ON IN RECIRC
   RUNG wire#powerrail
      Contact( "AlwaysTRUE" )
      { S7_Templates := "SrcType := Int" } EQ_Contact(in1 := "MODE SELECTION DB"."RO-1"."MODE BUFF", in2 := 1)
      { S7_Templates := "SrcType := Int" } EQ_Contact(in1 := "MODE SELECTION DB"."RO-1"."PROCESS BUFF", in2 := 2)
      { S7_Templates := "SrcType := Int" } EQ_Contact(in1 := "RO 1 LEVEL DB"."LEVEL HI RECIRC BUFF", in2 := 3)
      Contact( "RO_1 DB".OUTPUT."RO-1 HPP-301B" )
      Coil( "RO_1 DB".OUTPUT."AGLV-302 RECIRC" )
   END_RUNG
   // the same network as SCL:
   "RO_1 DB".OUTPUT."AGLV-302 RECIRC" := "AlwaysTRUE" AND ("MODE SELECTION DB"."RO-1"."MODE BUFF" = 1) AND ("MODE SELECTION DB"."RO-1"."PROCESS BUFF" = 2) AND ("RO 1 LEVEL DB"."LEVEL HI RECIRC BUFF" = 3) AND "RO_1 DB".OUTPUT."RO-1 HPP-301B";
END_REGION
END_FUNCTION
